TYPE ref_sv_output :
STRUCT
	out_flg_svA:	BOOL;
	out_flg_svB:	BOOL;
END_STRUCT
END_TYPE

(* stored: Version 1.1.0.1, ProductVersion 3.1.4024.11
   DUT ref_sv_output: Id {8ca9f649-156c-4f50-a557-38b188e6134b} *)
